Fanuc KAREL source: kb00068.KL

-- PROVISIONAL review KL for V770-1; original PC SHA256 1e9469254cda12501a93fa5f10af17881dea16dad4d9624b08db904a5011eafb
-- Incomplete behavior may be omitted. Consult companion uncertainty JSON. Do not deploy.
PROGRAM KB00068
%NOLOCKGROUP
BEGIN
  -- UNRESOLVED_PC offsets 5-14; opcodes 3F,75
  -- UNRESOLVED_PC offsets 19-26; opcodes 9D,23
  -- UNRESOLVED_PC offsets 31-49; opcodes 27,22,2A,22,31
  -- UNRESOLVED_PC offsets 54-58; opcodes 7F
END KB00068
